(* CoDeSys 2.3 library: OPC_error_AC500.lib *)
(* Libraries: SysLibRtc.lib 22.10.12 12:06:49, SysLibTime.lib 11.1.13 14:46:09, Standard.LIB 11.1.13 14:46:09 *)

(* Global variable list: OPC_Errors_Exchange *)
VAR_GLOBAL
	OpcExchange: OPC_ERROR;
	iNewOpcErr:INT;
	OPCLinkItem : UDINT := 0;	    (* notwendig für OPCServerLink*)
	HistUpdateCount: UDINT := 0;	(* notwendig für zyklischen Historyupdate*)
    ErrCrossCheck: UDINT := 0;      (* Gegenprüfung von Visu ob Fehler noch ansteht *)
    ErrCrossAck: UDINT := 0;        (* Bestaetigung von PLC ob Fehler noch ansteht *)
END_VAR

(* Global variable list: OPCErrors_Global *)
VAR_GLOBAL
	OpcErrFifo: ARRAY[0..255] OF OPC_ERROR;
	bOpcErrFifoWrIndex: BYTE;
	bOpcErrFifoRdIndex: BYTE;
	bOpcErrFifoCount:BYTE;
END_VAR

(* Data type *)
TYPE OPC_ERROR :
STRUCT
	Fault: INT;
	ArriveLeave: BOOL;
	tDateTime: DT;			(* yyyy mm dd hh mm ss*)
	MilliSeconds: DINT; (* msec *)
(*	ErrSubCode:INT;	(*used for CAN and IBS errors*)
	ErrSubType:INT;	(*used for CAN and IBS errors*)
	IbsSegment:INT;	(*used for IBS errors*)
	IbsPosition:INT;	(*used for IBS errors*)		*)
END_STRUCT
END_TYPE

(* POU OPC_ERR, ST *)
PROGRAM OPC_ERR
VAR_OUTPUT
END_VAR
VAR
	OldiOpcError: INT := -1;
END_VAR
(* letzter Fehler wurde bereits vom OPC-Client abgeholt *)
IF  ( iNewOpcErr <> OldiOpcError) THEN
	IF(bOpcErrFifoCount>0) THEN
		OpcExchange := OpcErrFifo[bOpcErrFifoRdIndex];
		bOpcErrFifoRdIndex := bOpcErrFifoRdIndex+1;
		bOpcErrFifoCount := bOpcErrFifoCount-1;
		(*gibt dem OpcClient an, dass ein neuer Fehler zum Abholen bereit steht *)
		iNewOpcErr :=iNewOpcErr + 1;
		OldiOpcError := iNewOpcErr;
	END_IF
END_IF
(* garantiert einen zyklischen Historyupdate *)
HistUpdateCount := HistUpdateCount + 1;
END_PROGRAM

(* POU ErrorClearToOpc, ST *)
FUNCTION ErrorClearToOpc:BOOL
VAR_INPUT
	Fault: INT;
	ErrSubCode:INT;	(*used for CAN and IBS errors*)
	ErrSubType:INT;	(*used for CAN and IBS errors*)
	IbsSegment:INT;	(*used for IBS errors*)
	IbsPosition:INT;	(*used for IBS errors*)
END_VAR
VAR
	OpcErr: OPC_ERROR;
END_VAR
OpcErr.Fault := Fault;
OpcErr.ArriveLeave := 0;
OpcErr.tDateTime := dtRead_Time;
OpcErr.MilliSeconds := 0;
(*OpcErr.ErrSubCode := ErrSubCode;	(*used for CAN and IBS errors*)
OpcErr.ErrSubType := ErrSubType;	(*used for CAN and IBS errors*)
OpcErr.IbsSegment :=  IbsSegment;	(*used for IBS errors*)
OpcErr.IbsPosition := IbsPosition;	(*used for IBS errors*)		*)
ErrorClearToOpc := OpcErrOutFifo(OpcErr);
END_FUNCTION

(* POU OpcErrOutFifo, ST *)
FUNCTION OpcErrOutFifo : BOOL
VAR_INPUT
	OpcErr: OPC_ERROR;
END_VAR
VAR
END_VAR
(* noch Platz im Fifo ?*)
IF(bOpcErrFifoCount<=255) THEN
	OpcErrFifo[bOpcErrFifoWrIndex] := OpcErr;
	bOpcErrFifoWrIndex := bOpcErrFifoWrIndex+1;
	bOpcErrFifoCount := bOpcErrFifoCount+1;
	OpcErrOutFifo:=TRUE;
ELSE
  OpcErrOutFifo:=FALSE;
END_IF
END_FUNCTION

(* POU ErrorSetToOpc, ST *)
FUNCTION ErrorSetToOpc:BOOL
VAR_INPUT
	Fault: INT;
	ErrSubCode:INT;	(*used for CAN and IBS errors*)
	ErrSubType:INT;	(*used for CAN and IBS errors*)
	IbsSegment:INT;	(*used for IBS errors*)
	IbsPosition:INT;	(*used for IBS errors*)
END_VAR
VAR
	OpcErr: OPC_ERROR;
END_VAR
OpcErr.Fault := Fault;
OpcErr.ArriveLeave := 1;
OpcErr.tDateTime := dtRead_Time;
OpcErr.MilliSeconds := 0;
(*OpcErr.ErrSubCode := ErrSubCode;	(*used for CAN and IBS errors*)
OpcErr.ErrSubType := ErrSubType;	(*used for CAN and IBS errors*)
OpcErr.IbsSegment :=  IbsSegment;	(*used for IBS errors*)
OpcErr.IbsPosition := IbsPosition;	(*used for IBS errors*)	*)
ErrorSetToOpc := OpcErrOutFifo(OpcErr);
END_FUNCTION

(* POU WarnClearToOpc, ST *)
FUNCTION WarnClearToOpc:BOOL
VAR_INPUT
	Fault: INT;
	ErrSubCode:INT;	(*used for CAN and IBS errors*)
	ErrSubType:INT;	(*used for CAN and IBS errors*)
	IbsSegment:INT;	(*used for IBS errors*)
	IbsPosition:INT;	(*used for IBS errors*)
END_VAR
VAR
	OpcErr: OPC_ERROR;
END_VAR
OpcErr.Fault := Fault;
OpcErr.ArriveLeave := 0;
OpcErr.tDateTime := dtRead_Time;
OpcErr.MilliSeconds := 0;
(*OpcErr.ErrSubCode := ErrSubCode;	(*used for CAN and IBS errors*)
OpcErr.ErrSubType := ErrSubType;	(*used for CAN and IBS errors*)
OpcErr.IbsSegment :=  IbsSegment;	(*used for IBS errors*)
OpcErr.IbsPosition := IbsPosition;	(*used for IBS errors*)		*)
WarnClearToOpc := OpcErrOutFifo(OpcErr);
END_FUNCTION

(* POU WarnSetToOpc, ST *)
FUNCTION WarnSetToOpc:BOOL
VAR_INPUT
	Fault: INT;
	ErrSubCode:INT;	(*used for CAN and IBS errors*)
	ErrSubType:INT;	(*used for CAN and IBS errors*)
	IbsSegment:INT;	(*used for IBS errors*)
	IbsPosition:INT;	(*used for IBS errors*)
END_VAR
VAR
	OpcErr: OPC_ERROR;
END_VAR
OpcErr.Fault := Fault;
OpcErr.ArriveLeave := 1;
OpcErr.tDateTime := dtRead_Time;
OpcErr.MilliSeconds := 0;
(*OpcErr.ErrSubCode := ErrSubCode;	(*used for CAN and IBS errors*)
OpcErr.ErrSubType := ErrSubType;	(*used for CAN and IBS errors*)
OpcErr.IbsSegment :=  IbsSegment;	(*used for IBS errors*)
OpcErr.IbsPosition := IbsPosition;	(*used for IBS errors*)		*)
WarnSetToOpc := OpcErrOutFifo(OpcErr);
END_FUNCTION
